(* Logix 5000 project; controller PBS_Perfusion vendor 1 type 14 code 217 rev 32.14; software revision 32.03; part 2 of 27 *)
(* tags used below, declared in another part *)
   ONS : DINT[3];
   REAL : DINT;

ADD_ON_INSTRUCTION AMP_Hard_Stop_Homing   (* revision 1.0 *)
// Applied Motion - Hard Stop Homing AOI
// Help:
// The Hard Stop Homing AOI accepts all the required parameters for SCL commands HV1, HV2, HV3, HA1, HA2, HA3, HL1, HL2, HL3, HC, HD, HO and then sends the HS command to initiate the Hard Stop Homing move.
VAR_IN_OUT
   Input : DINT[14]; {required}   // Drive Input Assembly
   Output : DINT[16]; {required}   // Drive Output Assembly
        [0]   // Command Word
        [1]   // Jog Speed (0.25 rev/min)
        [2]   // Jog Acceleration (10 rev/s/s)
        [3]   // Jog Deceleration (10 rev/s/s)
        [4]   // Point-to-Point Velocity (0.25 rev/min)
        [5]   // Point-to-Point Acceleration (10 rev/s/s)
        [6]   // Point-to-Point Deceleration (10 rev/s/s)
        [7]   // Point-to-Point Distance (Motor steps)
        [9]   // (2x ASCII Letters in 16 lower word)
        [10]   // Data/Register 1
        [11]   // Data/Register 2
END_VAR
VAR_INPUT
   RPI : DINT := 100; {visible}   // Drive Connection Request Packet Interval (milliseconds)
   Start : BOOL; {required}   // Start the Homing
   HV1 : REAL; {required}   // Velocity used while seeking the hard stop (rev/s)
   HV2 : REAL; {required}   // Velocity when moving offset distance set by HO (rev/s)
   HV3 : REAL; {required}   // Velocity when searching for encoder index if desired (rev/s)
   HA1 : REAL; {required}   // Accel used while seeking the hard stop (rev/s/s)
   HA2 : REAL; {required}   // Accel when moving offset distance set by HO (rev/s/s)
   HA3 : REAL; {required}   // Accel when searching for encoder index if desired (rev/s/s)
   HL1 : REAL; {required}   // Decel used while seeking the hard stop (rev/s/s)
   HL2 : REAL; {required}   // Decel when moving offset distance set by HO (rev/s/s)
   HL3 : REAL; {required}   // Decel when searching for encoder index if desired (rev/s/s)
   HC : REAL; {required}   // Hard Stop Current (Amps)
   HD : DINT; {required}   // Hard Stop Fault Delay (ms)
   HO : DINT; {required}   // Home Offset (steps, negative = CCW, positive = CW)
   HS : DINT; {required}   // Hard Stop method (0 = without index, 1 = with index)
END_VAR
VAR_OUTPUT
   Sent : BOOL; {access Read Only, visible}   // All parameter setting and homing commands have been sent to drive
   In_Progress : BOOL; {access Read Only, visible}   // The setting of parameters and/or homing are in progress
   Done : BOOL; {access Read Only, visible}   // Homing Move completed without errors - desired position reached
   Error : BOOL; {access Read Only, visible}   // Homing failed to complete - drive not ready or faulted
   State : DINT := 34; {access Read Only}   // Internal state of progress
END_VAR
VAR
   Loc_StatusCode : AMP_Status_Word;
   Loc_CommandOff_Timer : TIMER;   // Timer to make sure command value was 0 before sending a new command
   Loc_CommandOn_Timer : TIMER;   // Timer to make sure command value is set long enough to be sent to drive
   Loc_Input_Assembly : AMP_Input_Assembly_v2; {access None}
   Loc_Start_ONS : BOOL; {access None}
END_VAR

ROUTINE Logic   (* ladder *)
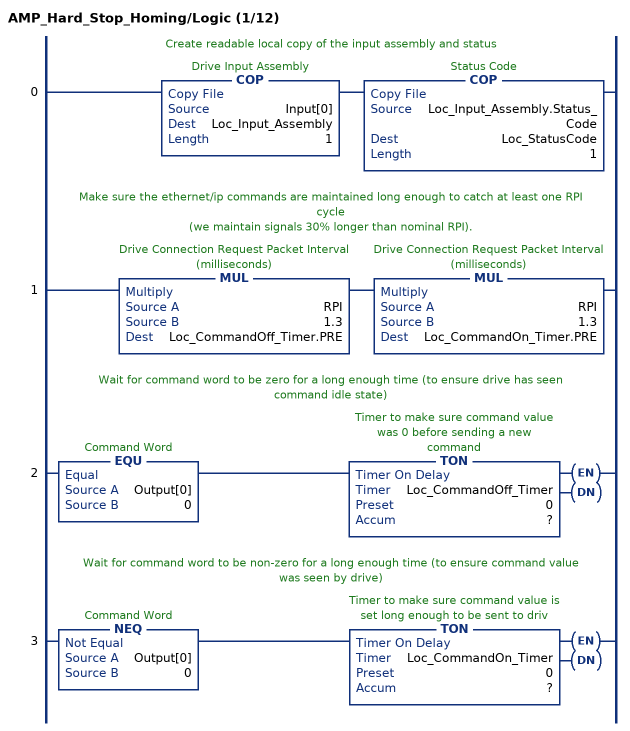
   // Create readable local copy of the input assembly and status
   0: COP(Input[0],Loc_Input_Assembly,1)COP(Loc_Input_Assembly.Status_Code,Loc_StatusCode,1);
   // Make sure the ethernet/ip commands are maintained long enough to catch at least one RPI cycle
   // (we maintain signals 30% longer than nominal RPI).
   1: MUL(RPI,1.3,Loc_CommandOff_Timer.PRE)MUL(RPI,1.3,Loc_CommandOn_Timer.PRE);
   // Wait for command word to be zero for a long enough time (to ensure drive has seen command idle state)
   2: EQU(Output[0],0)TON(Loc_CommandOff_Timer,?,?);
   // Wait for command word to be non-zero for a long enough time (to ensure command value was seen by drive)
   3: NEQ(Output[0],0)TON(Loc_CommandOn_Timer,?,?);
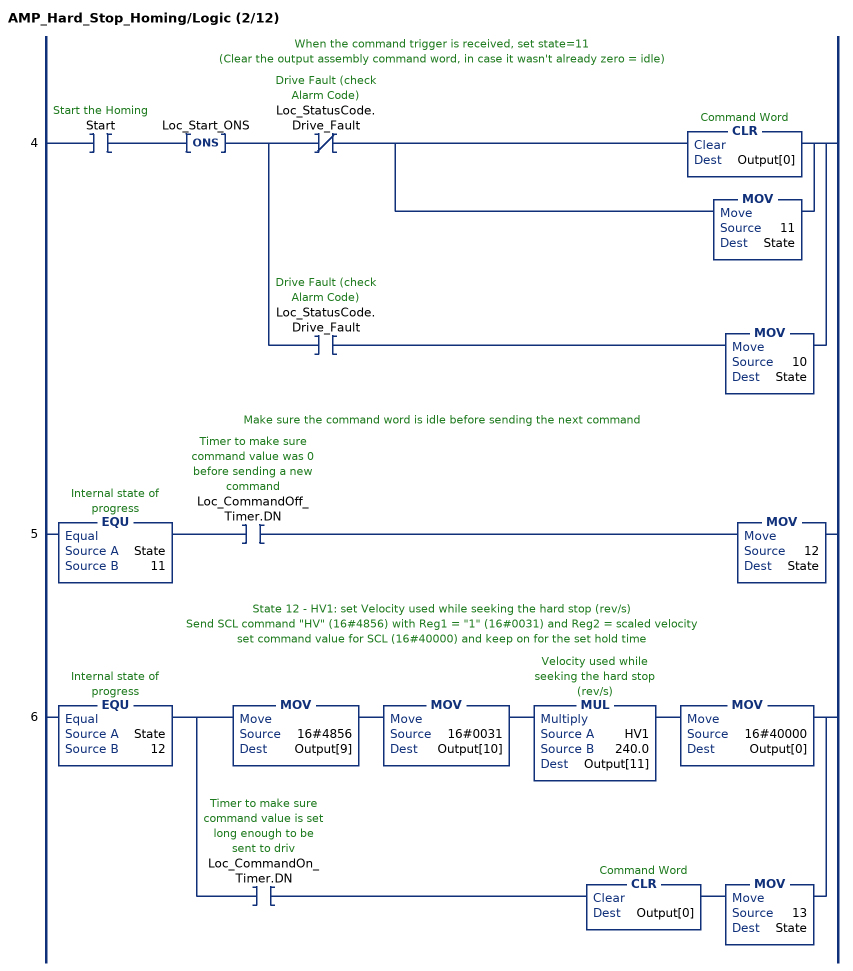
   // When the command trigger is received, set state=11
   // (Clear the output assembly command word, in case it wasn't already zero = idle)
   4: XIC(Start)ONS(Loc_Start_ONS)[XIO(Loc_StatusCode.Drive_Fault) [CLR(Output[0]) ,MOV(11,State) ] ,XIC(Loc_StatusCode.Drive_Fault) MOV(10,State) ];
   // Make sure the command word is idle before sending the next command
   5: EQU(State,11)XIC(Loc_CommandOff_Timer.DN)MOV(12,State);
   // State 12 - HV1: set Velocity used while seeking the hard stop (rev/s)
   // Send SCL command "HV" (16#4856) with Reg1 = "1" (16#0031) and Reg2 = scaled velocity
   // set command value for SCL (16#40000) and keep on for the set hold time
   6: EQU(State,12)[MOV(16#4856,Output[9]) MOV(16#0031,Output[10]) MUL(HV1,240.0,Output[11]) MOV(16#40000,Output[0]) ,XIC(Loc_CommandOn_Timer.DN) CLR(Output[0]) MOV(13,State) ];
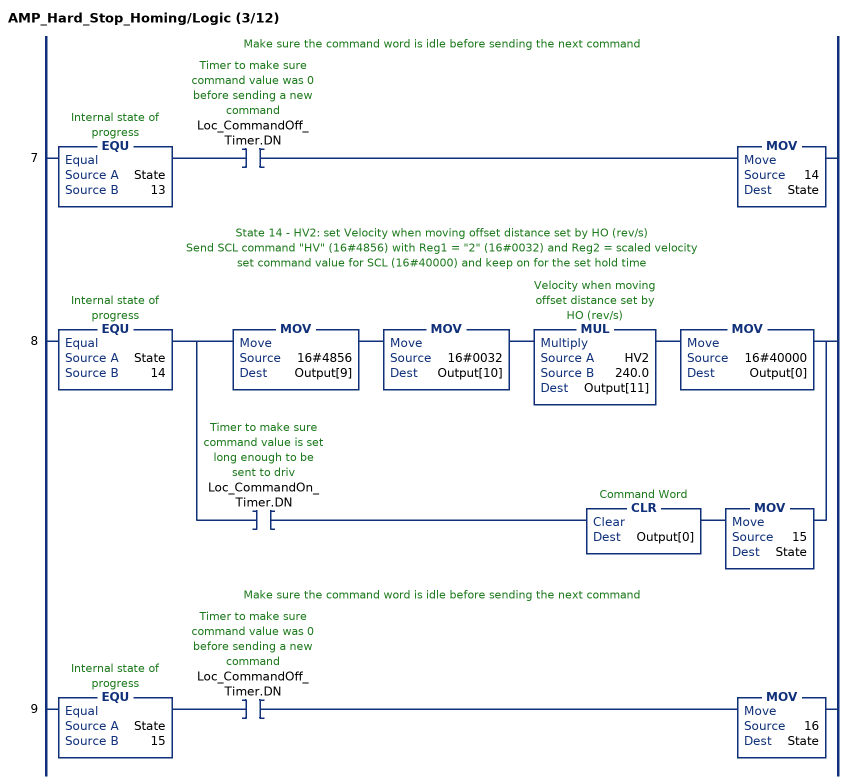
   // Make sure the command word is idle before sending the next command
   7: EQU(State,13)XIC(Loc_CommandOff_Timer.DN)MOV(14,State);
   // State 14 - HV2: set Velocity when moving offset distance set by HO (rev/s)
   // Send SCL command "HV" (16#4856) with Reg1 = "2" (16#0032) and Reg2 = scaled velocity
   // set command value for SCL (16#40000) and keep on for the set hold time
   8: EQU(State,14)[MOV(16#4856,Output[9]) MOV(16#0032,Output[10]) MUL(HV2,240.0,Output[11]) MOV(16#40000,Output[0]) ,XIC(Loc_CommandOn_Timer.DN) CLR(Output[0]) MOV(15,State) ];
   // Make sure the command word is idle before sending the next command
   9: EQU(State,15)XIC(Loc_CommandOff_Timer.DN)MOV(16,State);
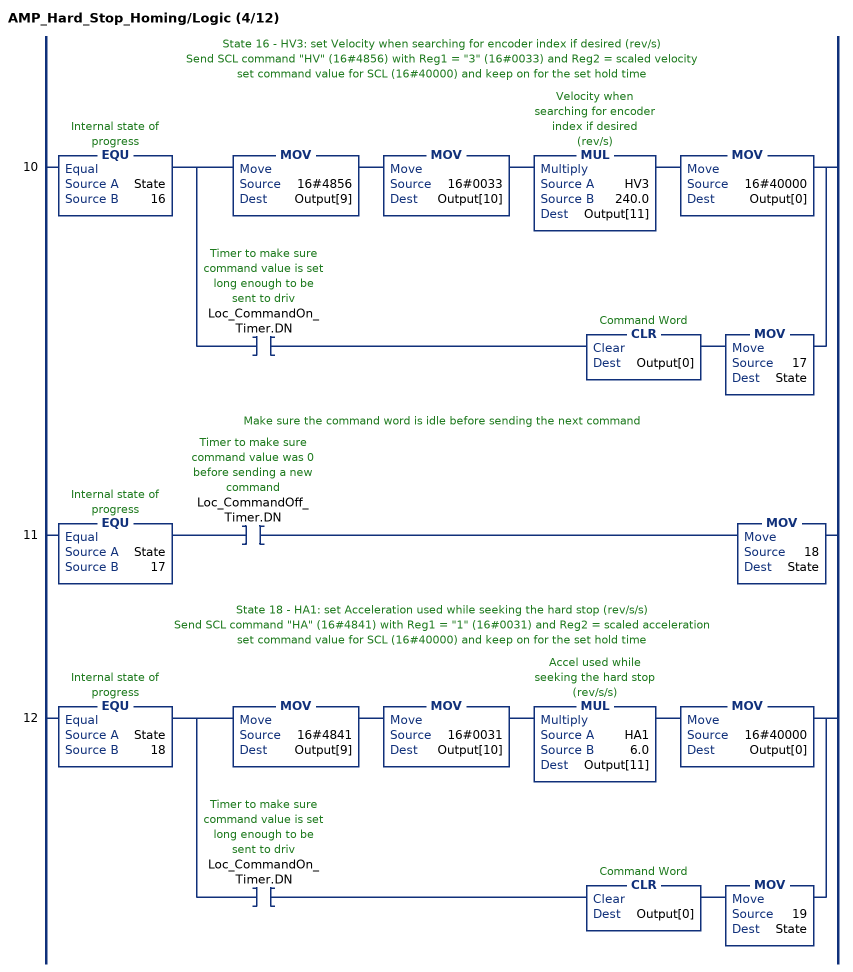
   // State 16 - HV3: set Velocity when searching for encoder index if desired (rev/s)
   // Send SCL command "HV" (16#4856) with Reg1 = "3" (16#0033) and Reg2 = scaled velocity
   // set command value for SCL (16#40000) and keep on for the set hold time
   10: EQU(State,16)[MOV(16#4856,Output[9]) MOV(16#0033,Output[10]) MUL(HV3,240.0,Output[11]) MOV(16#40000,Output[0]) ,XIC(Loc_CommandOn_Timer.DN) CLR(Output[0]) MOV(17,State) ];
   // Make sure the command word is idle before sending the next command
   11: EQU(State,17)XIC(Loc_CommandOff_Timer.DN)MOV(18,State);
   // State 18 - HA1: set Acceleration used while seeking the hard stop (rev/s/s)
   // Send SCL command "HA" (16#4841) with Reg1 = "1" (16#0031) and Reg2 = scaled acceleration
   // set command value for SCL (16#40000) and keep on for the set hold time
   12: EQU(State,18)[MOV(16#4841,Output[9]) MOV(16#0031,Output[10]) MUL(HA1,6.0,Output[11]) MOV(16#40000,Output[0]) ,XIC(Loc_CommandOn_Timer.DN) CLR(Output[0]) MOV(19,State) ];
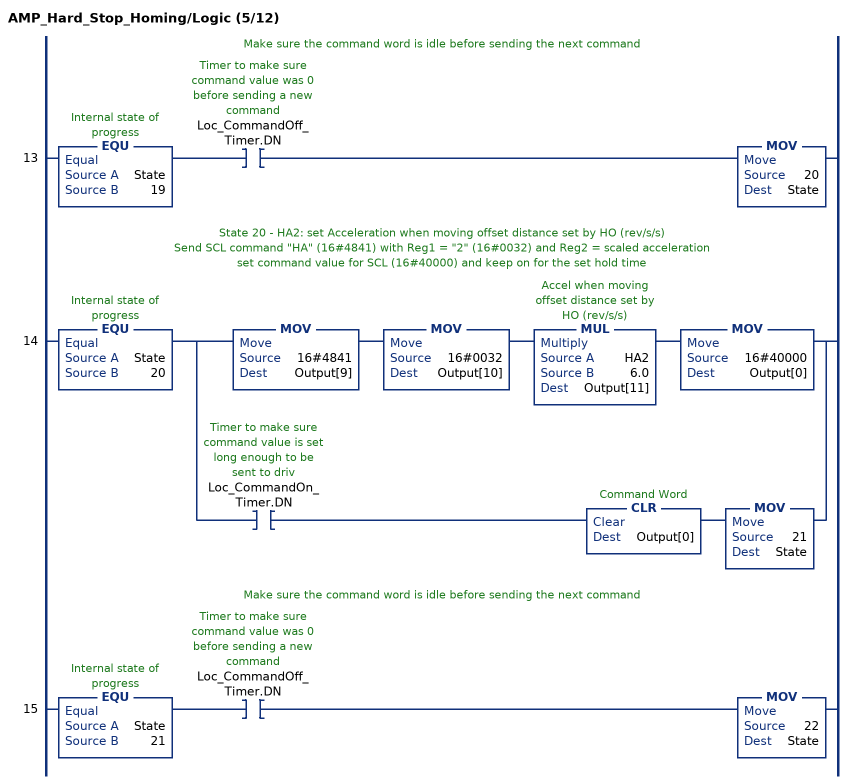
   // Make sure the command word is idle before sending the next command
   13: EQU(State,19)XIC(Loc_CommandOff_Timer.DN)MOV(20,State);
   // State 20 - HA2: set Acceleration when moving offset distance set by HO (rev/s/s)
   // Send SCL command "HA" (16#4841) with Reg1 = "2" (16#0032) and Reg2 = scaled acceleration
   // set command value for SCL (16#40000) and keep on for the set hold time
   14: EQU(State,20)[MOV(16#4841,Output[9]) MOV(16#0032,Output[10]) MUL(HA2,6.0,Output[11]) MOV(16#40000,Output[0]) ,XIC(Loc_CommandOn_Timer.DN) CLR(Output[0]) MOV(21,State) ];
   // Make sure the command word is idle before sending the next command
   15: EQU(State,21)XIC(Loc_CommandOff_Timer.DN)MOV(22,State);
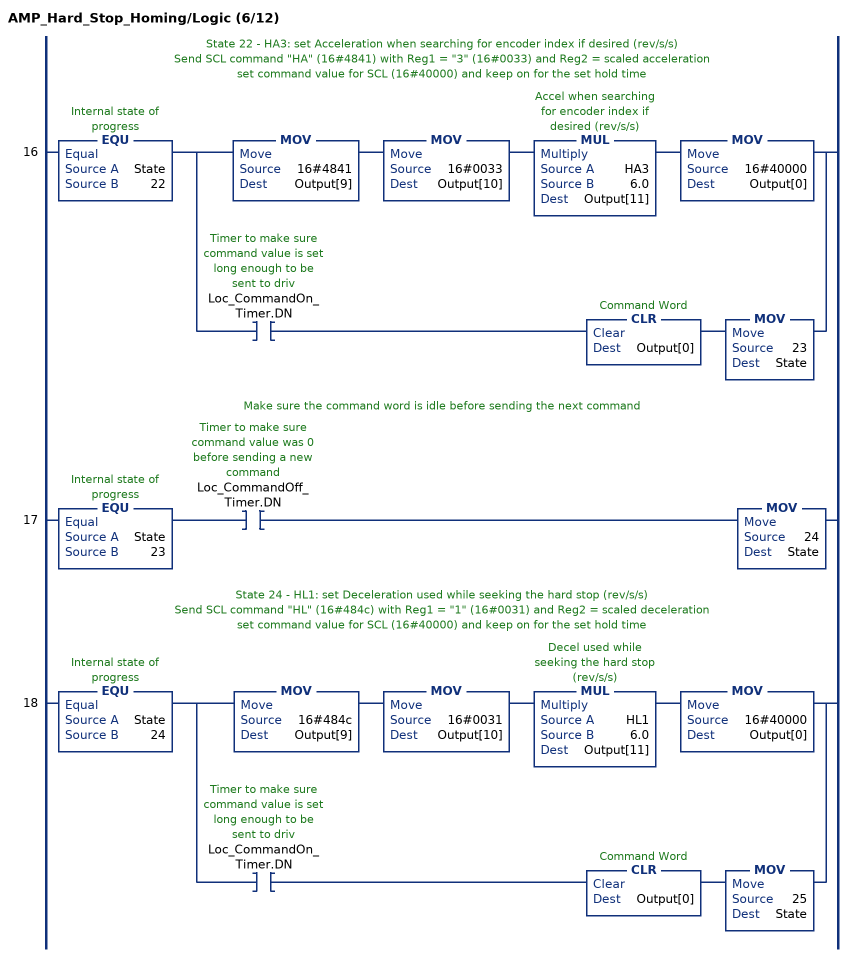
   // State 22 - HA3: set Acceleration when searching for encoder index if desired (rev/s/s)
   // Send SCL command "HA" (16#4841) with Reg1 = "3" (16#0033) and Reg2 = scaled acceleration
   // set command value for SCL (16#40000) and keep on for the set hold time
   16: EQU(State,22)[MOV(16#4841,Output[9]) MOV(16#0033,Output[10]) MUL(HA3,6.0,Output[11]) MOV(16#40000,Output[0]) ,XIC(Loc_CommandOn_Timer.DN) CLR(Output[0]) MOV(23,State) ];
   // Make sure the command word is idle before sending the next command
   17: EQU(State,23)XIC(Loc_CommandOff_Timer.DN)MOV(24,State);
   // State 24 - HL1: set Deceleration used while seeking the hard stop (rev/s/s)
   // Send SCL command "HL" (16#484c) with Reg1 = "1" (16#0031) and Reg2 = scaled deceleration
   // set command value for SCL (16#40000) and keep on for the set hold time
   18: EQU(State,24)[MOV(16#484c,Output[9]) MOV(16#0031,Output[10]) MUL(HL1,6.0,Output[11]) MOV(16#40000,Output[0]) ,XIC(Loc_CommandOn_Timer.DN) CLR(Output[0]) MOV(25,State) ];
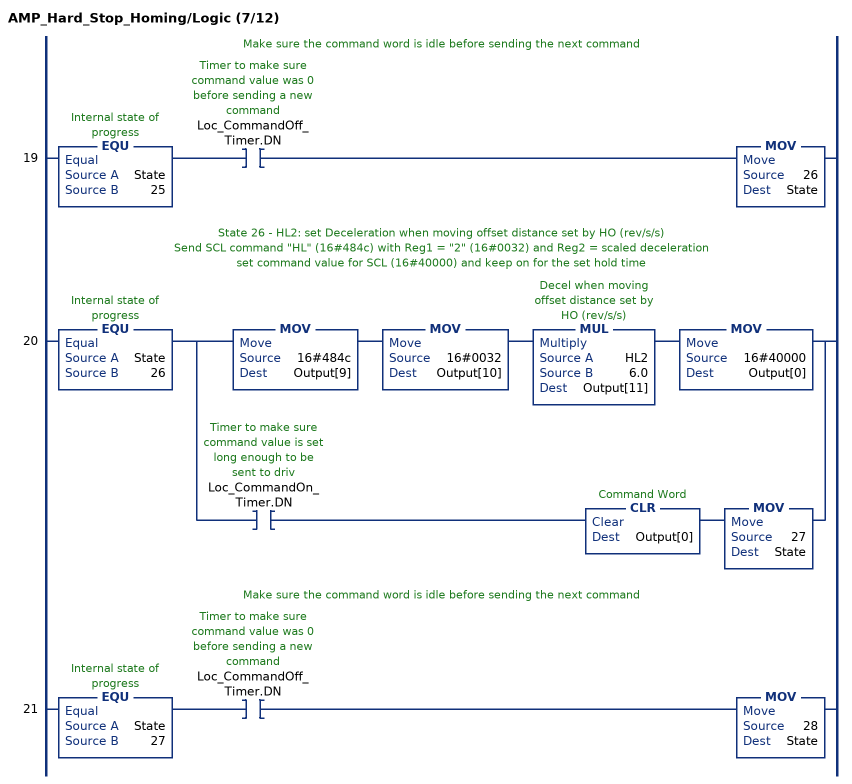
   // Make sure the command word is idle before sending the next command
   19: EQU(State,25)XIC(Loc_CommandOff_Timer.DN)MOV(26,State);
   // State 26 - HL2: set Deceleration when moving offset distance set by HO (rev/s/s)
   // Send SCL command "HL" (16#484c) with Reg1 = "2" (16#0032) and Reg2 = scaled deceleration
   // set command value for SCL (16#40000) and keep on for the set hold time
   20: EQU(State,26)[MOV(16#484c,Output[9]) MOV(16#0032,Output[10]) MUL(HL2,6.0,Output[11]) MOV(16#40000,Output[0]) ,XIC(Loc_CommandOn_Timer.DN) CLR(Output[0]) MOV(27,State) ];
   // Make sure the command word is idle before sending the next command
   21: EQU(State,27)XIC(Loc_CommandOff_Timer.DN)MOV(28,State);
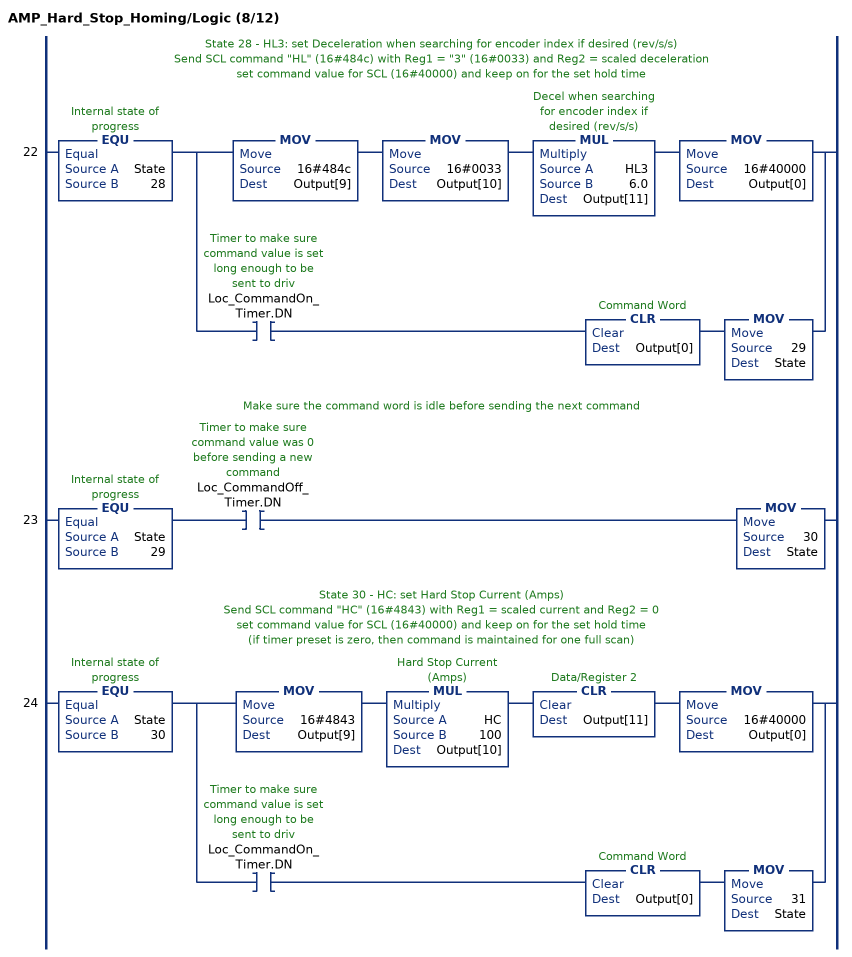
   // State 28 - HL3: set Deceleration when searching for encoder index if desired (rev/s/s)
   // Send SCL command "HL" (16#484c) with Reg1 = "3" (16#0033) and Reg2 = scaled deceleration
   // set command value for SCL (16#40000) and keep on for the set hold time
   22: EQU(State,28)[MOV(16#484c,Output[9]) MOV(16#0033,Output[10]) MUL(HL3,6.0,Output[11]) MOV(16#40000,Output[0]) ,XIC(Loc_CommandOn_Timer.DN) CLR(Output[0]) MOV(29,State) ];
   // Make sure the command word is idle before sending the next command
   23: EQU(State,29)XIC(Loc_CommandOff_Timer.DN)MOV(30,State);
   // State 30 - HC: set Hard Stop Current (Amps)
   // Send SCL command "HC" (16#4843) with Reg1 = scaled current and Reg2 = 0
   // set command value for SCL (16#40000) and keep on for the set hold time
   // (if timer preset is zero, then command is maintained for one full scan)
   24: EQU(State,30)[MOV(16#4843,Output[9]) MUL(HC,100,Output[10]) CLR(Output[11]) MOV(16#40000,Output[0]) ,XIC(Loc_CommandOn_Timer.DN) CLR(Output[0]) MOV(31,State) ];
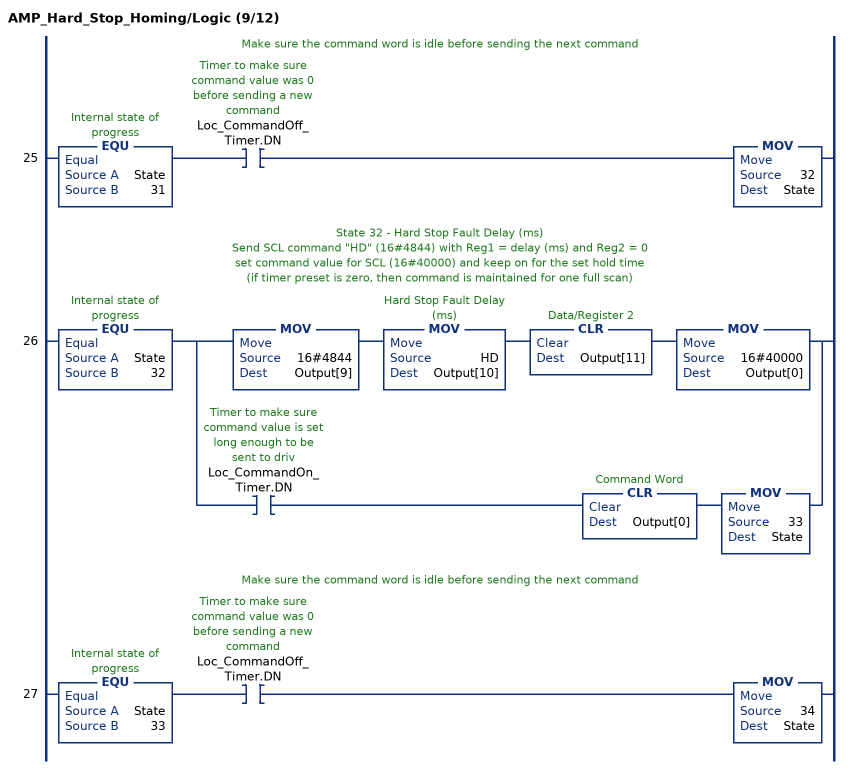
   // Make sure the command word is idle before sending the next command
   25: EQU(State,31)XIC(Loc_CommandOff_Timer.DN)MOV(32,State);
   // State 32 - Hard Stop Fault Delay (ms)
   // Send SCL command "HD" (16#4844) with Reg1 = delay (ms) and Reg2 = 0
   // set command value for SCL (16#40000) and keep on for the set hold time
   // (if timer preset is zero, then command is maintained for one full scan)
   26: EQU(State,32)[MOV(16#4844,Output[9]) MOV(HD,Output[10]) CLR(Output[11]) MOV(16#40000,Output[0]) ,XIC(Loc_CommandOn_Timer.DN) CLR(Output[0]) MOV(33,State) ];
   // Make sure the command word is idle before sending the next command
   27: EQU(State,33)XIC(Loc_CommandOff_Timer.DN)MOV(34,State);
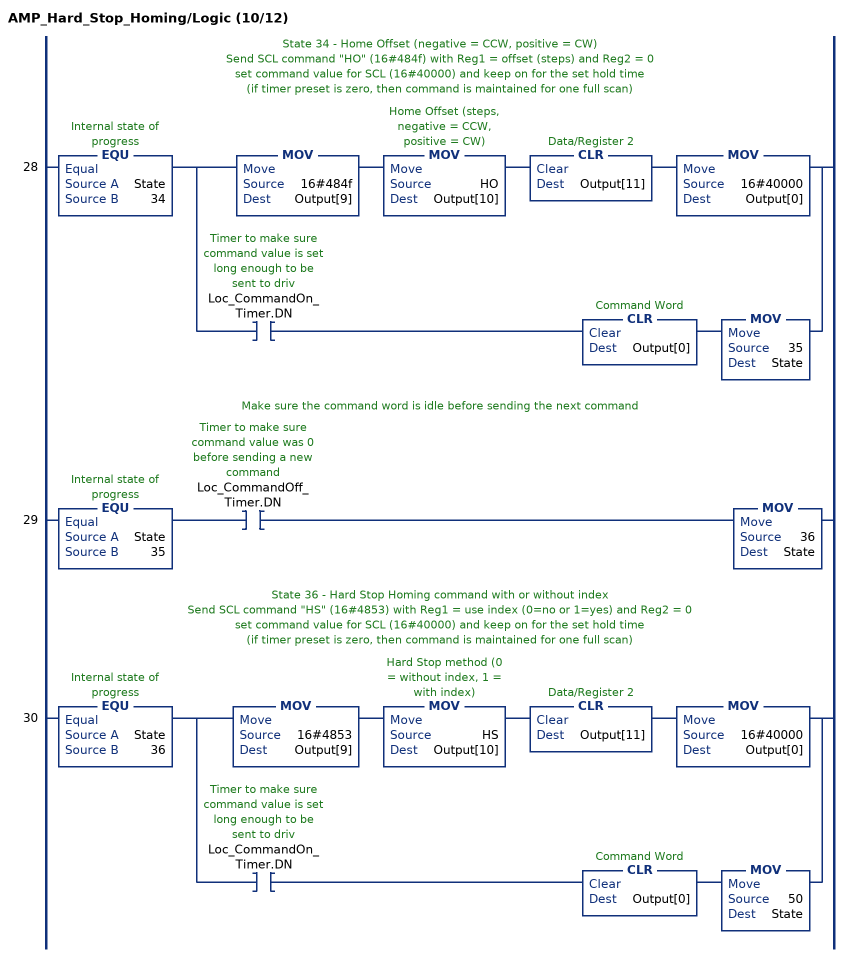
   // State 34 - Home Offset (negative = CCW, positive = CW)
   // Send SCL command "HO" (16#484f) with Reg1 = offset (steps) and Reg2 = 0
   // set command value for SCL (16#40000) and keep on for the set hold time
   // (if timer preset is zero, then command is maintained for one full scan)
   28: EQU(State,34)[MOV(16#484f,Output[9]) MOV(HO,Output[10]) CLR(Output[11]) MOV(16#40000,Output[0]) ,XIC(Loc_CommandOn_Timer.DN) CLR(Output[0]) MOV(35,State) ];
   // Make sure the command word is idle before sending the next command
   29: EQU(State,35)XIC(Loc_CommandOff_Timer.DN)MOV(36,State);
   // State 36 - Hard Stop Homing command with or without index
   // Send SCL command "HS" (16#4853) with Reg1 = use index (0=no or 1=yes) and Reg2 = 0
   // set command value for SCL (16#40000) and keep on for the set hold time
   // (if timer preset is zero, then command is maintained for one full scan)
   30: EQU(State,36)[MOV(16#4853,Output[9]) MOV(HS,Output[10]) CLR(Output[11]) MOV(16#40000,Output[0]) ,XIC(Loc_CommandOn_Timer.DN) CLR(Output[0]) MOV(50,State) ];
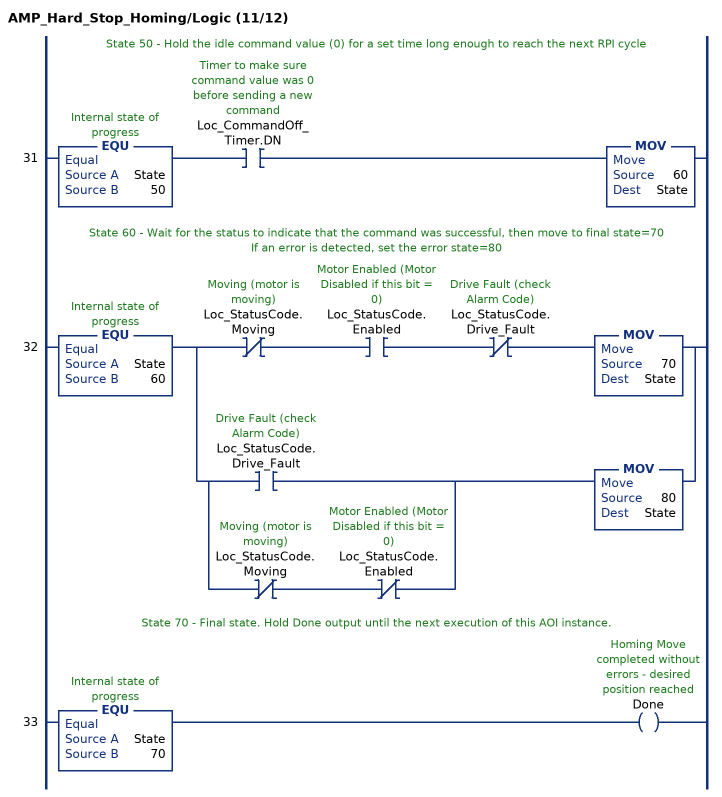
   // State 50 - Hold the idle command value (0) for a set time long enough to reach the next RPI cycle
   31: EQU(State,50)XIC(Loc_CommandOff_Timer.DN)MOV(60,State);
   // State 60 - Wait for the status to indicate that the command was successful, then move to final state=70
   // If an error is detected, set the error state=80
   32: EQU(State,60)[XIO(Loc_StatusCode.Moving) XIC(Loc_StatusCode.Enabled) XIO(Loc_StatusCode.Drive_Fault) MOV(70,State) ,[XIC(Loc_StatusCode.Drive_Fault) ,XIO(Loc_StatusCode.Moving) XIO(Loc_StatusCode.Enabled) ] MOV(80,State) ];
   // State 70 - Final state. Hold Done output until the next execution of this AOI instance.
   33: EQU(State,70)OTE(Done);
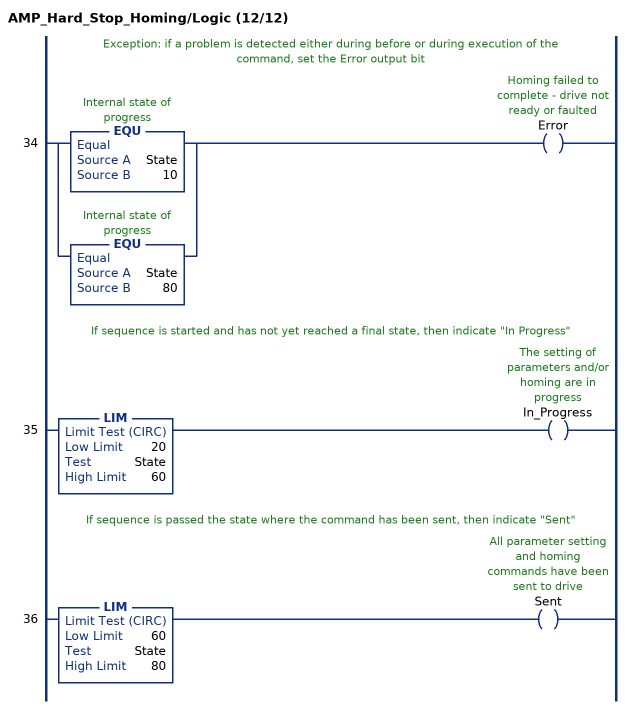
   // Exception: if a problem is detected either during before or during execution of the command, set the Error output bit
   34: [EQU(State,10) ,EQU(State,80) ]OTE(Error);
   // If sequence is started and has not yet reached a final state, then indicate "In Progress"
   35: LIM(20,State,60)OTE(In_Progress);
   // If sequence is passed the state where the command has been sent, then indicate "Sent"
   36: LIM(60,State,80)OTE(Sent);
END_ROUTINE
END_ADD_ON_INSTRUCTION

ADD_ON_INSTRUCTION AMP_Input_Assembly   (* revision 1.0 *)
// Applied Motion - Input Assembly AOI
// Help:
// The Input Assembly AOI takes raw input data from the drive and re-interprets the data, using either scaling or copying, to appropriately named outputs.
VAR_IN_OUT
   Input : DINT[14]; {required}   // AMP_Assembly
   Output : AMP_Input_Assembly_v2; {required}
END_VAR
VAR_OUTPUT
   Status_Code : DINT; {access Read Only, visible}   // Status Code
   Alarm_Code : DINT; {access Read Only, visible}   // Alarm Code
   Voltage : REAL; {access Read Only, visible}   // Supply Voltage (V)
   Current : REAL; {access Read Only, visible}   // Actual Current (mA)
   Temp : REAL; {access Read Only, visible}   // Drive Temperature (deg C)
   Encoder_Position : DINT; {access Read Only, visible}   // Encoder Position (20,000 counts = 1 shaft turn)
   Absolute_Position : DINT; {access Read Only, visible}   // Absolute Position (20,000 counts = 1 shaft turn)
   Actual_Velocity : REAL; {access Read Only, visible}   // Actual Velocity (rev/sec, 0 when no encoder)
   Position_Error : DINT; {access Read Only, visible}
   Extended_Inputs : INT; {access Read Only, visible}   // Input Status (Extended)
   Main_Board_Inputs : INT; {access Read Only, visible}   // Input Status (Main board)
   Analog_Input_1 : DINT; {access Read Only, visible}   // Analog Input 1 (ADC counts, 0=min V, 16383 = max V)
   Analog_Input_2 : DINT; {access Read Only, visible}   // Analog Input 2 (ADC counts, 0=min V, 16383 = max V)
END_VAR
VAR
   Loc_Input_Assembly : AMP_Input_Assembly_v2; {access None}
   Loc_StatusCode : AMP_Status_Word; {access None}
END_VAR

ROUTINE Logic   (* ladder *)
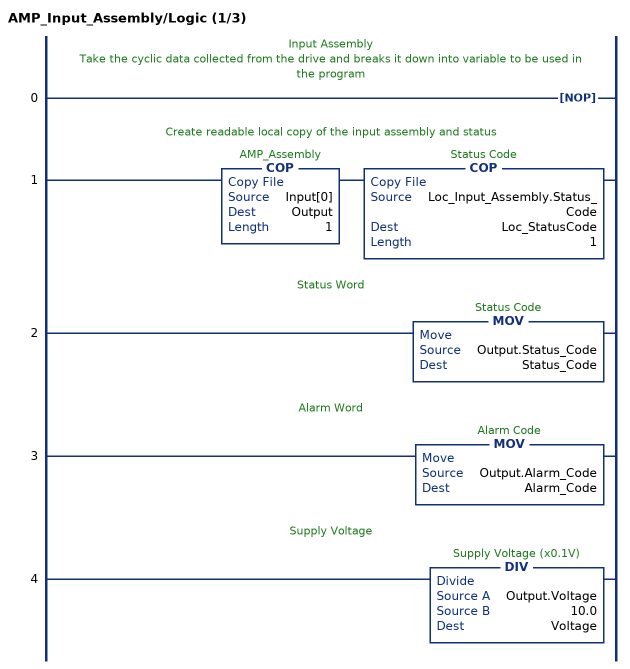
   // Input Assembly
   // Take the cyclic data collected from the drive and breaks it down into variable to be used in the program
   0: NOP();
   // Create readable local copy of the input assembly and status
   1: COP(Input[0],Output,1)COP(Loc_Input_Assembly.Status_Code,Loc_StatusCode,1);
   // Status Word
   2: MOV(Output.Status_Code,Status_Code);
   // Alarm Word
   3: MOV(Output.Alarm_Code,Alarm_Code);
   // Supply Voltage
   4: DIV(Output.Voltage,10.0,Voltage);
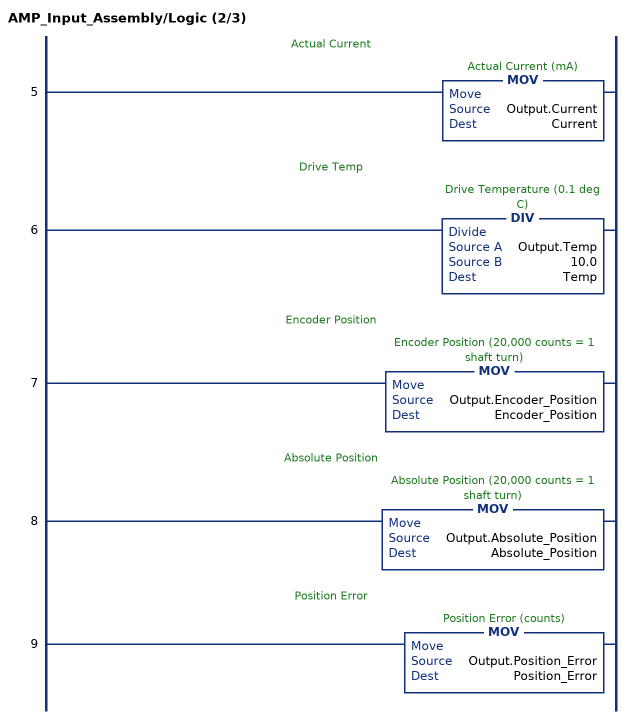
   // Actual Current
   5: MOV(Output.Current,Current);
   // Drive Temp
   6: DIV(Output.Temp,10.0,Temp);
   // Encoder Position
   7: MOV(Output.Encoder_Position,Encoder_Position);
   // Absolute Position
   8: MOV(Output.Absolute_Position,Absolute_Position);
   // Position Error
   9: MOV(Output.Position_Error,Position_Error);
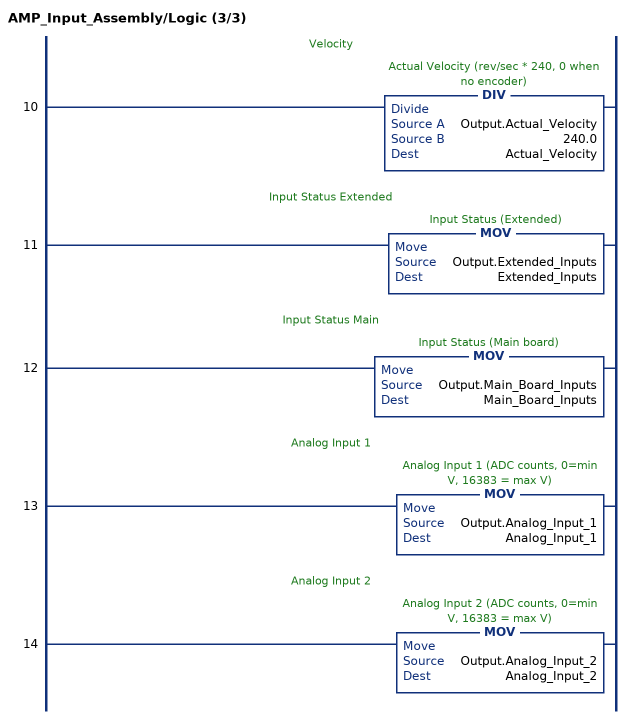
   // Velocity
   10: DIV(Output.Actual_Velocity,240.0,Actual_Velocity);
   // Input Status Extended
   11: MOV(Output.Extended_Inputs,Extended_Inputs);
   // Input Status Main
   12: MOV(Output.Main_Board_Inputs,Main_Board_Inputs);
   // Analog Input 1
   13: MOV(Output.Analog_Input_1,Analog_Input_1);
   // Analog Input 2
   14: MOV(Output.Analog_Input_2,Analog_Input_2);
END_ROUTINE
END_ADD_ON_INSTRUCTION

ADD_ON_INSTRUCTION AMP_Jog_Move   (* revision 1.0 *)
// Applied Motion - Jog Move AOI
// Help:
// The Jog Move AOI is used to start jogging an axis at a specified speed and direction (a negative speed set point implies a CCW direction).
VAR_IN_OUT
   Input : DINT[14]; {required}   // Drive Input Assembly
   Output : DINT[16]; {required}   // Drive Output Assembly
        [0]   // Command Word
        [1]   // Jog Speed (0.25 rev/min)
        [2]   // Jog Acceleration (10 rev/s/s)
        [3]   // Jog Deceleration (10 rev/s/s)
        [4]   // Point-to-Point Velocity (0.25 rev/min)
        [5]   // Point-to-Point Acceleration (10 rev/min/s)
        [6]   // Point-to-Point Deceleration (10 rev/min/s)
        [7]   // Point-to-Point Distance (Motor steps)
        [9]   // (2x ASCII Letters in 16 lower word)
        [10]   // Data/Register 1
        [11]   // Data/Register 2
END_VAR
VAR_INPUT
   RPI : DINT := 100; {visible}   // Drive Connection Request Packet Interval (milliseconds)
   Start : BOOL; {required}   // Start the Relative Move
   Speed : REAL; {required}   // Velocity of Move (rev/min)
   Acc : REAL; {required}   // Acceleration of Move (rev/s/s)
   Dec : REAL; {required}   // Deceleration (rev/s/s)
END_VAR
VAR_OUTPUT
   Sent : BOOL; {access Read Only, visible}   // Move has been sent to drive
   In_Progress : BOOL; {access Read Only, visible}   // Move in progress
   Done : BOOL; {access Read Only, visible}   // Move completed without errors - desired position reached
   Error : BOOL; {access Read Only, visible}   // Move failed to complete - drive not ready or faulted
   State : DINT := 10; {access Read Only}   // Internal state of progress
END_VAR
VAR
   Loc_StatusCode : AMP_Status_Word;
   Loc_CommandOff_Timer : TIMER;   // Timer to make sure command value was 0 before sending a new command
   Loc_CommandOn_Timer : TIMER;   // Timer to make sure command value is set long enough to be sent to drive
   Loc_Input_Assembly : AMP_Input_Assembly_v2; {access None}
   Loc_Start_ONS : BOOL; {access None}
   Loc_AlarmCode : AMP_Alarm_Word; {access None}
END_VAR

ROUTINE Logic   (* ladder *)
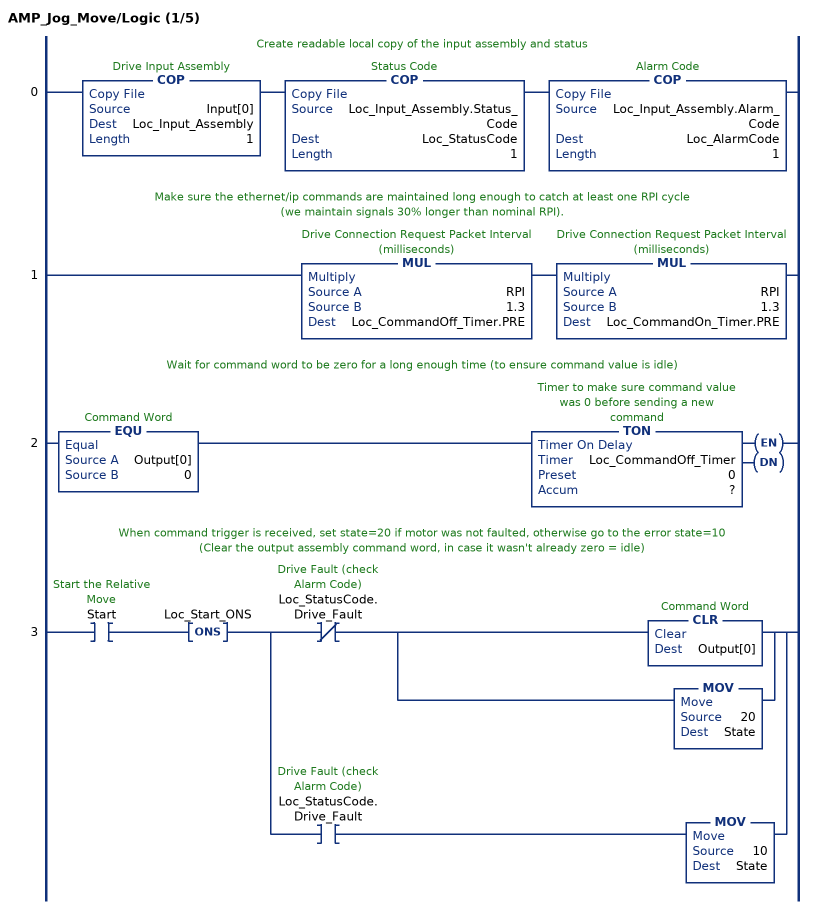
   // Create readable local copy of the input assembly and status
   0: COP(Input[0],Loc_Input_Assembly,1)COP(Loc_Input_Assembly.Status_Code,Loc_StatusCode,1)COP(Loc_Input_Assembly.Alarm_Code,Loc_AlarmCode,1);
   // Make sure the ethernet/ip commands are maintained long enough to catch at least one RPI cycle
   // (we maintain signals 30% longer than nominal RPI).
   1: MUL(RPI,1.3,Loc_CommandOff_Timer.PRE)MUL(RPI,1.3,Loc_CommandOn_Timer.PRE);
   // Wait for command word to be zero for a long enough time (to ensure command value is idle)
   2: EQU(Output[0],0)TON(Loc_CommandOff_Timer,?,?);
   // When command trigger is received, set state=20 if motor was not faulted, otherwise go to the error state=10
   // (Clear the output assembly command word, in case it wasn't already zero = idle)
   3: XIC(Start)ONS(Loc_Start_ONS)[XIO(Loc_StatusCode.Drive_Fault) [CLR(Output[0]) ,MOV(20,State) ] ,XIC(Loc_StatusCode.Drive_Fault) MOV(10,State) ];
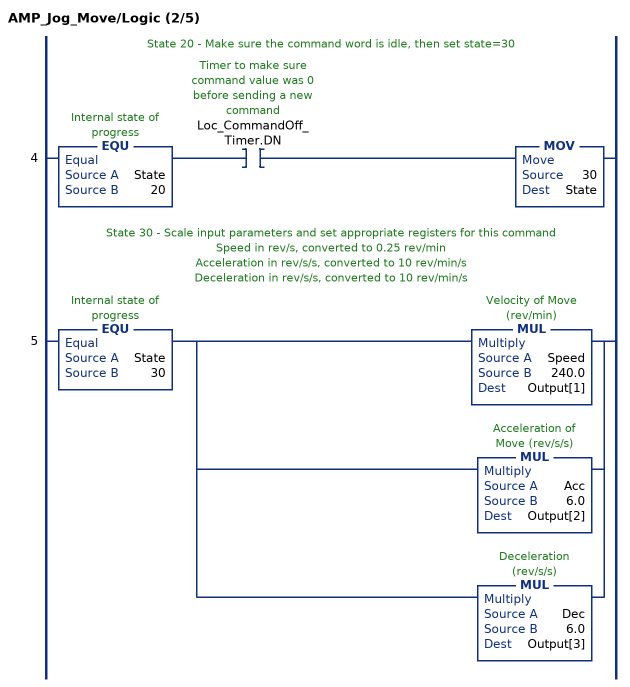
   // State 20 - Make sure the command word is idle, then set state=30
   4: EQU(State,20)XIC(Loc_CommandOff_Timer.DN)MOV(30,State);
   // State 30 - Scale input parameters and set appropriate registers for this command
   // Speed in rev/s, converted to 0.25 rev/min
   // Acceleration in rev/s/s, converted to 10 rev/min/s
   // Deceleration in rev/s/s, converted to 10 rev/min/s
   5: EQU(State,30)[MUL(Speed,240.0,Output[1]) ,MUL(Acc,6.0,Output[2]) ,MUL(Dec,6.0,Output[3]) ];
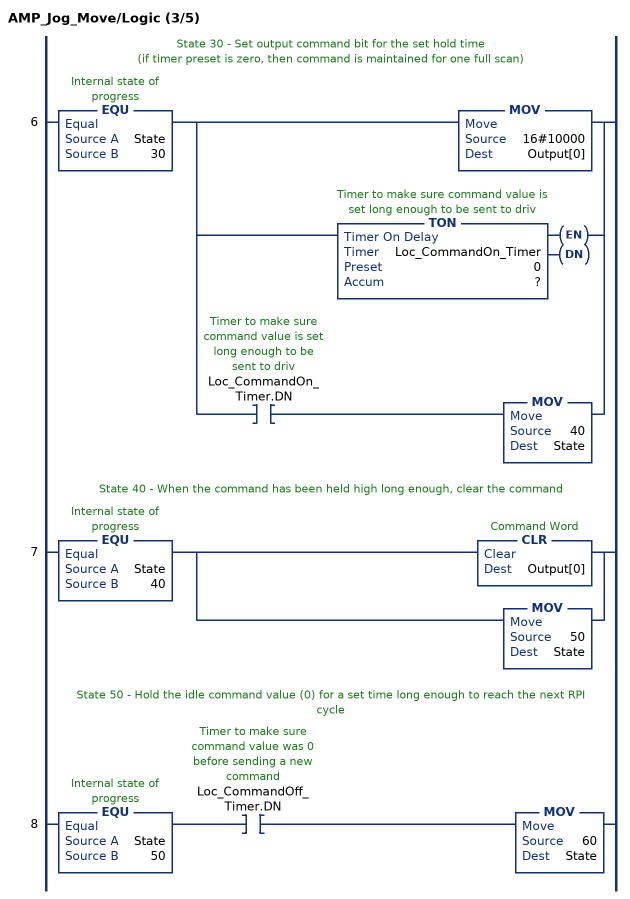
   // State 30 - Set output command bit for the set hold time
   // (if timer preset is zero, then command is maintained for one full scan)
   6: EQU(State,30)[MOV(16#10000,Output[0]) ,TON(Loc_CommandOn_Timer,?,?) ,XIC(Loc_CommandOn_Timer.DN) MOV(40,State) ];
   // State 40 - When the command has been held high long enough, clear the command
   7: EQU(State,40)[CLR(Output[0]) ,MOV(50,State) ];
   // State 50 - Hold the idle command value (0) for a set time long enough to reach the next RPI cycle
   8: EQU(State,50)XIC(Loc_CommandOff_Timer.DN)MOV(60,State);
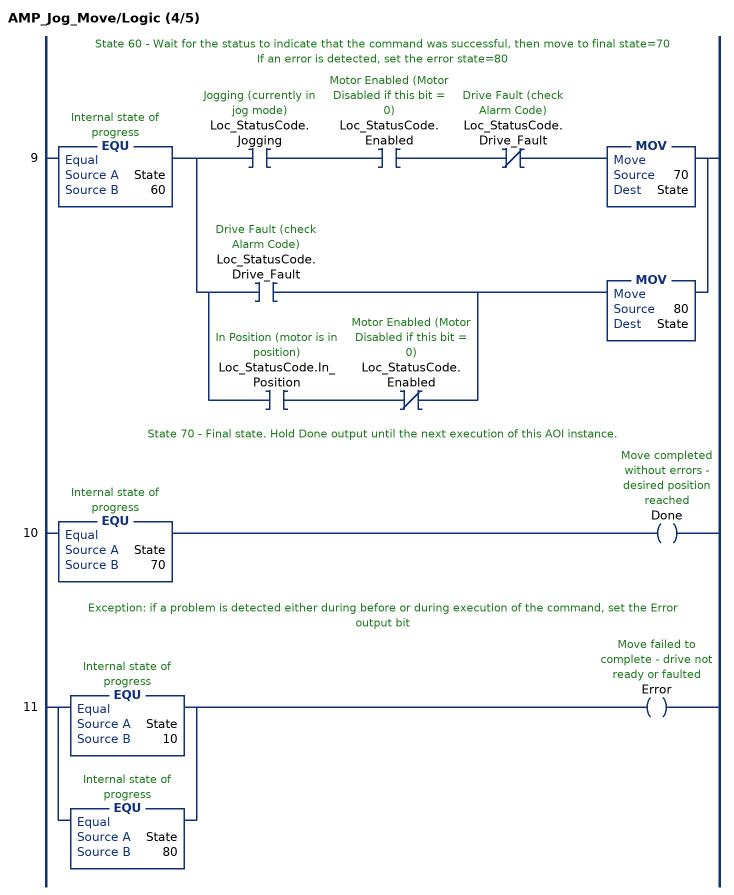
   // State 60 - Wait for the status to indicate that the command was successful, then move to final state=70
   // If an error is detected, set the error state=80
   9: EQU(State,60)[XIC(Loc_StatusCode.Jogging) XIC(Loc_StatusCode.Enabled) XIO(Loc_StatusCode.Drive_Fault) MOV(70,State) ,[XIC(Loc_StatusCode.Drive_Fault) ,XIC(Loc_StatusCode.In_Position) XIO(Loc_StatusCode.Enabled) ] MOV(80,State) ];
   // State 70 - Final state. Hold Done output until the next execution of this AOI instance.
   10: EQU(State,70)OTE(Done);
   // Exception: if a problem is detected either during before or during execution of the command, set the Error output bit
   11: [EQU(State,10) ,EQU(State,80) ]OTE(Error);
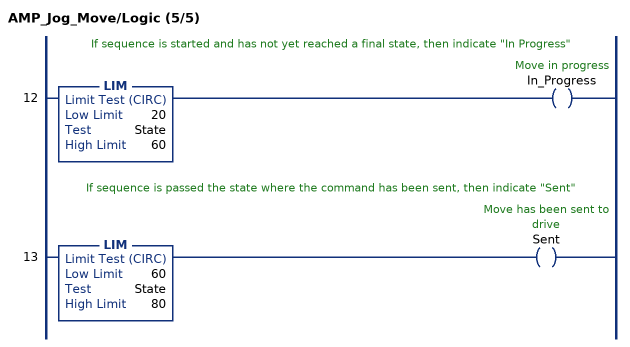
   // If sequence is started and has not yet reached a final state, then indicate "In Progress"
   12: LIM(20,State,60)OTE(In_Progress);
   // If sequence is passed the state where the command has been sent, then indicate "Sent"
   13: LIM(60,State,80)OTE(Sent);
END_ROUTINE
END_ADD_ON_INSTRUCTION
